FUNCTION_BLOCK Kullager
  (* Version 0.1, 2005-04-08, Kobetski Flordal, Chalmers *)
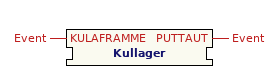
  EVENT_INPUT
    KULAFRAMME;
  END_EVENT
  EVENT_OUTPUT
    PUTTAUT;
  END_EVENT
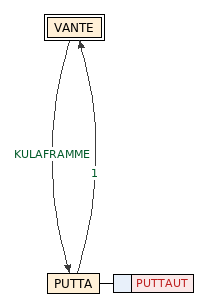
  EC_STATES
    VANTE;
    PUTTA : -> PUTTAUT;
  END_STATES
  EC_TRANSITIONS
    VANTE TO PUTTA := KULAFRAMME;
    PUTTA TO VANTE := 1;
  END_TRANSITIONS
END_FUNCTION_BLOCK
